FUNCTION_BLOCK "Net"
{ S7_Optimized_Access := 'TRUE' }
AUTHOR : Searinox
VERSION : 0.1
   VAR_INPUT
      iAutoMode : Bool;
      iPumpPlant1 : "Pump";
      iPumpPlant2 : "Pump";
      iPumpCoolWater1 : "Pump";
      iPumpCoolWater2 : "Pump";
      iPumpFurnace1 : "Pump";
      iPumpFurnace2 : "Pump";
      iFan1 : "Fan";
      iFan2 : "Fan";
      iSprayPipe1 : "Valve";
      iSprayPipe2 : "Valve";
      iSurgeTankRefill : "Valve";
      iLiftingSys1 : "LiftingSys";
      iLiftingSys2 : "LiftingSys";
      iTempPlant : "Temperature";
      iTempFurnace : "Temperature";
      iSurgeTank : "Tank";
      iBleedingUnit : "BleedingUnit";
   END_VAR

   VAR_IN_OUT
      ioAlarm : "Alarm";
   END_VAR

   VAR
      sAlarmCount : Int;
      sAlarmCountCrit : Int;
      sAlarms : Struct
         Crit : Struct
            CvOff : Int;
            FuseOutputsErr : Int;
            FanErrCrit : Int;
            PumpPlantErrCrit : Int;
            PumpCoolWaterErrCrit : Int;
            PumpFurnaceErrCrit : Int;
            SurgeTankRunDry : Int;
            SurgeTankOverflow : Int;
         END_STRUCT;
         Ct1FanErr : Int;
         Ct1RepairSwitchOff : Int;
         Ct2FanErr : Int;
         Ct2RepairSwitchOff : Int;
         PumpPlant1Err : Int;
         PumpPlant2Err : Int;
         PumpCoolWater1Err : Int;
         PumpCoolWater2Err : Int;
         PumpFurnace1Err : Int;
         PumpFurnace2Err : Int;
         FlowTempPlantHot : Int;
         FlowTempFurnaceHot : Int;
         PressureDeltaPerc1 : Int;
         PressureDeltaPerc2 : Int;
         SprayPipeOpenTimeout1 : Int;
         SprayPipeOpenTimeout2 : Int;
         BleedingUnitErr : Int;
      END_STRUCT;
      sAutoMode : Bool;
      sPumpPlant1 : Struct
         Q : Bool;
         IsRunning : Bool;
         HasError : Bool;
      END_STRUCT;
      sPumpPlant2 : Struct
         Q : Bool;
         IsRunning : Bool;
         HasError : Bool;
      END_STRUCT;
      sPumpCoolWater1 : Struct
         Q : Bool;
         IsRunning : Bool;
         HasError : Bool;
      END_STRUCT;
      sPumpCoolWater2 : Struct
         Q : Bool;
         IsRunning : Bool;
         HasError : Bool;
      END_STRUCT;
      sPumpFurnace1 : Struct
         Q : Bool;
         IsRunning : Bool;
         HasError : Bool;
      END_STRUCT;
      sPumpFurnace2 : Struct
         Q : Bool;
         IsRunning : Bool;
         HasError : Bool;
      END_STRUCT;
      sFan1 : Struct
         Q : Bool;
         IsRunning : Bool;
         HasError : Bool;
         RepairSwitch : Bool;
         SetPoint : Int;
      END_STRUCT;
      sFan2 : Struct
         Q : Bool;
         IsRunning : Bool;
         HasError : Bool;
         RepairSwitch : Bool;
         SetPoint : Int;
      END_STRUCT;
      sSprayPipe1 : Struct
         Q : Bool;
         IsOpen : Bool;
         Timeout : Time;
      END_STRUCT;
      sSprayPipe2 : Struct
         Q : Bool;
         IsOpen : Bool;
         Timeout : Time;
      END_STRUCT;
      sSurgeTankRefill : Struct
         Q : Bool;
         IsOpen : Bool;
         IsClosed : Bool;
         HasError : Bool;
         SetPoint : Int;
         Timeout : Time;
      END_STRUCT;
      sLiftingSys1 : Struct
         DeltaPressure : Struct
            IW : Int;
            Val : Real;
            Limits : Struct
               Min : Real;
               Max : Real;
            END_STRUCT;
         END_STRUCT;
      END_STRUCT;
      sLiftingSys2 : Struct
         DeltaPressure : Struct
            IW : Int;
            Val : Real;
            Limits : Struct
               Min : Real;
               Max : Real;
            END_STRUCT;
         END_STRUCT;
      END_STRUCT;
      sTempPlant : Struct
         IW : Int;
         Val : Real;
         Limits : Struct
            Min : Real;
            Max : Real;
         END_STRUCT;
      END_STRUCT;
      sTempFurnace : Struct
         IW : Int;
         Val : Real;
         Limits : Struct
            Min : Real;
            Max : Real;
         END_STRUCT;
      END_STRUCT;
      sSurgeTank : Struct
         Val : Int;
         Levels : Struct
            RunDry : Int;
            SetPointLower : Int;
            SetPointUpper : Int;
            Overflow : Int;
         END_STRUCT;
      END_STRUCT;
      sBleedingUnit : Struct
         IsRunning : Bool;
         HasError : Bool;
      END_STRUCT;
   END_VAR


BEGIN
	#sAlarmCount := #ioAlarm.oAlarmCount;
	#sAlarmCountCrit := #ioAlarm.oAlarmCountCrit;
	#sAlarms.BleedingUnitErr := #ioAlarm.sBleedingUnitErr;
	#sAlarms.Crit.CvOff := #ioAlarm.sCvOff;
	#sAlarms.Crit.FanErrCrit := #ioAlarm.sFanErrCrit;
	#sAlarms.Crit.FuseOutputsErr := #ioAlarm.sFuseOutputsErr;
	#sAlarms.Crit.PumpCoolWaterErrCrit := #ioAlarm.sPumpCoolWaterErrCrit;
	#sAlarms.Crit.PumpFurnaceErrCrit := #ioAlarm.sPumpFurnaceErrCrit;
	#sAlarms.Crit.PumpPlantErrCrit := #ioAlarm.sPumpPlantErrCrit;
	#sAlarms.Crit.SurgeTankOverflow := #ioAlarm.sSurgeTankOverflow;
	#sAlarms.Crit.SurgeTankRunDry := #ioAlarm.sSurgeTankRunDry;
	#sAlarms.Ct1FanErr := #ioAlarm.sCt1FanErr;
	#sAlarms.Ct1RepairSwitchOff := #ioAlarm.sCt1RepairSwitchOff;
	#sAlarms.Ct2FanErr := #ioAlarm.sCt2FanErr;
	#sAlarms.Ct2RepairSwitchOff := #ioAlarm.sCt2RepairSwitchOff;
	#sAlarms.FlowTempFurnaceHot := #ioAlarm.sFlowTempFurnaceHot;
	#sAlarms.FlowTempPlantHot := #ioAlarm.sFlowTempPlantHot;
	#sAlarms.PressureDeltaPerc1 := #ioAlarm.sPressureDeltaPerc1;
	#sAlarms.PressureDeltaPerc2 := #ioAlarm.sPressureDeltaPerc2;
	#sAlarms.PumpCoolWater1Err := #ioAlarm.sPumpCoolWater1Err;
	#sAlarms.PumpCoolWater2Err := #ioAlarm.sPumpCoolWater2Err;
	#sAlarms.PumpFurnace1Err := #ioAlarm.sPumpFurnace1Err;
	#sAlarms.PumpFurnace2Err := #ioAlarm.sPumpFurnace2Err;
	#sAlarms.PumpPlant1Err := #ioAlarm.sPumpPlant1Err;
	#sAlarms.PumpPlant2Err := #ioAlarm.sPumpPlant2Err;
	#sAlarms.SprayPipeOpenTimeout1 := #ioAlarm.sSprayPipeOpenTimeout1;
	#sAlarms.SprayPipeOpenTimeout2 := #ioAlarm.sSprayPipeOpenTimeout2;
	#sAutoMode := #iAutoMode;
	#sBleedingUnit.HasError := #iBleedingUnit.HasError;
	#sBleedingUnit.IsRunning := #iBleedingUnit.IsRunning;
	#sFan1.HasError := #iFan1.HasError;
	#sFan1.IsRunning := #iFan1.IsRunning;
	#sFan1.Q := #iFan1.Q;
	#sFan1.RepairSwitch := #iFan1.RepairSwitch;
	#sFan1.SetPoint := #iFan1.SetPoint;
	#sFan2.HasError := #iFan2.HasError;
	#sFan2.IsRunning := #iFan2.IsRunning;
	#sFan2.Q := #iFan2.Q;
	#sFan2.RepairSwitch := #iFan2.RepairSwitch;
	#sFan2.SetPoint := #iFan2.SetPoint;
	#sLiftingSys1.DeltaPressure.IW := #iLiftingSys1.DeltaPressure.IW;
	#sLiftingSys1.DeltaPressure.Limits.Max := #iLiftingSys1.DeltaPressure.Limits.Max.R;
	#sLiftingSys1.DeltaPressure.Limits.Min := #iLiftingSys1.DeltaPressure.Limits.Min.R;
	#sLiftingSys1.DeltaPressure.Val := #iLiftingSys1.DeltaPressure.Val.R;
	#sLiftingSys2.DeltaPressure.IW := #iLiftingSys2.DeltaPressure.IW;
	#sLiftingSys2.DeltaPressure.Limits.Max := #iLiftingSys2.DeltaPressure.Limits.Max.R;
	#sLiftingSys2.DeltaPressure.Limits.Min := #iLiftingSys2.DeltaPressure.Limits.Min.R;
	#sLiftingSys2.DeltaPressure.Val := #iLiftingSys2.DeltaPressure.Val.R;
	#sPumpCoolWater1.HasError := #iPumpCoolWater1.HasError;
	#sPumpCoolWater1.IsRunning := #iPumpCoolWater1.IsRunning;
	#sPumpCoolWater1.Q := #iPumpCoolWater1.Q;
	#sPumpCoolWater2.HasError := #iPumpCoolWater2.HasError;
	#sPumpCoolWater2.IsRunning := #iPumpCoolWater2.IsRunning;
	#sPumpCoolWater2.Q := #iPumpCoolWater2.Q;
	#sPumpFurnace1.HasError := #iPumpFurnace1.HasError;
	#sPumpFurnace1.IsRunning := #iPumpFurnace1.IsRunning;
	#sPumpFurnace1.Q := #iPumpFurnace1.Q;
	#sPumpFurnace2.HasError := #iPumpFurnace2.HasError;
	#sPumpFurnace2.IsRunning := #iPumpFurnace2.IsRunning;
	#sPumpFurnace2.Q := #iPumpFurnace2.Q;
	#sPumpPlant1.HasError := #iPumpPlant1.HasError;
	#sPumpPlant1.IsRunning := #iPumpPlant1.IsRunning;
	#sPumpPlant1.Q := #iPumpPlant1.Q;
	#sPumpPlant2.HasError := #iPumpPlant2.HasError;
	#sPumpPlant2.IsRunning := #iPumpPlant2.IsRunning;
	#sPumpPlant2.Q := #iPumpPlant2.Q;
	#sSprayPipe1.IsOpen := #iSprayPipe1.IsOpen;
	#sSprayPipe1.Q := #iSprayPipe1.Q;
	#sSprayPipe1.Timeout := #iSprayPipe1.Timeout;
	#sSprayPipe2.IsOpen := #iSprayPipe2.IsOpen;
	#sSprayPipe2.Q := #iSprayPipe2.Q;
	#sSprayPipe2.Timeout := #iSprayPipe2.Timeout;
	#sSurgeTank.Levels.Overflow := #iSurgeTank.Levels.Overflow;
	#sSurgeTank.Levels.RunDry := #iSurgeTank.Levels.RunDry;
	#sSurgeTank.Levels.SetPointLower := #iSurgeTank.Levels.SetPointLower;
	#sSurgeTank.Levels.SetPointUpper := #iSurgeTank.Levels.SetPointUpper;
	#sSurgeTank.Val := #iSurgeTank.Val.I;
	#sSurgeTankRefill.Q := #iSurgeTankRefill.Q;
	#sSurgeTankRefill.IsOpen := #iSurgeTankRefill.IsOpen;
	#sTempFurnace.IW := #iTempFurnace.IW;
	#sTempFurnace.Limits.Max := #iTempFurnace.Limits.Max.R;
	#sTempFurnace.Limits.Min := #iTempFurnace.Limits.Min.R;
	#sTempFurnace.Val := #iTempFurnace.Val.R;
	#sTempPlant.IW := #iTempPlant.IW;
	#sTempPlant.Limits.Max := #iTempPlant.Limits.Max.R;
	#sTempPlant.Limits.Min := #iTempPlant.Limits.Min.R;
	#sTempPlant.Val := #iTempPlant.Val.R;

END_FUNCTION_BLOCK

